TEXTLIST TextList_07
  0 = 'Wybierz język' | pl: 'Wybierz język' | en: 'Select language' | de: 'Sprache auswählen'
  1 = 'Utwórz szablon receptur' | pl: 'Utwórz szablon receptur' | en: 'Create a recipe template' | de: 'Erstellen Sie eine Rezeptvorlage'
  2 = 'Utworzenie szablonów spowoduje usunięcie istniejących receptur' | pl: 'Utworzenie szablonów spowoduje usunięcie istniejących receptur' | en: 'Creating templates will delete existing recipes' | de: 'Beim Erstellen von Vorlagen werden bestehende Rezepte gelöscht.'
  3 = 'Utwórz' | pl: 'Utwórz' | en: 'Create' | de: 'Erstellen'
   = ''
END_TEXTLIST

(* stored: Version 1.1.0.1
   TextList TextList_07: Id {98639942-4805-0e52-29b6-cbef38307b96} *)
